(* Logix 5000 project; controller Comas_L4 vendor 1 type 14 code 193 rev 30.11; software revision 30.02; part 10 of 12 *)
(* tags used below, declared in another part *)
   Activation_Rouleau : BOOL;
   Axe_Codeur_Four : AXIS_CIP_DRIVE;
   Axe_Coupe_Fil : AXIS_CIP_DRIVE;
   Axe_Rouleaux_Canneles : AXIS_CIP_DRIVE;
   Axe_Virtuel_Coupe_Fil : AXIS_VIRTUAL;
   Axe_Virtuel_Maitre : AXIS_VIRTUAL;
   Cadencement_Moyennage_Codeur : FBD_TIMER;
   CAM_Virtuel_Coupe_Fil : CAM[100];
   CamGenerator_Coupe_Fil : AOI_CamGenerator_ST;
   CF_Mode_Came_Activation : BOOL;
   CF_Mode_Came_Engagement : BOOL;
   CF_Mode_Top_Activation : BOOL;
   CF_Mode_Top_Mouvement : BOOL;
   CO_Acquit_defaut : BOOL;
   CO_Activation : BOOL;
   CO_Axe_Codeur_Four_OK : BOOL;
   CO_Axe_Coupe_Fil_OK : BOOL;
   CO_Axe_Horizontal_Droit_OK : BOOL;
   CO_Axe_Horizontal_Gauche_OK : BOOL;
   CO_Axe_Pompe_Doseuse_OK : BOOL;
   CO_Axe_Rouleaux_Canneles_OK : BOOL;
   CO_Axe_Vertical_Droit_OK : BOOL;
   CO_Axe_Vertical_Gauche_OK : BOOL;
   CO_Consigne_Vitesse_Rouleaux : REAL;
   CO_Defaut_ARU_Armoire : BOOL;
   CO_Defaut_ARU_Machine : BOOL;
   CO_Defaut_ARU_Pupitre : BOOL;
   CO_Defaut_CamGenerator_Coupe_Fil : BOOL;
   CO_Defaut_CamGenerator_Horizontal : BOOL;
   CO_Defaut_CamGenerator_Vertical : BOOL;
   CO_Defaut_Clef_Graissage : BOOL;
   CO_Defaut_CPT_Porte1 : BOOL;
   CO_Defaut_CPT_Porte2 : BOOL;
   CO_Defaut_CPT_Porte3 : BOOL;
   CO_Defaut_CPT_Porte4 : BOOL;
   CO_Defaut_Eth_Codeur_Four : BOOL;
   CO_Defaut_Eth_Var_Coupe_Fil : BOOL;
   CO_Defaut_Eth_Var_H_Droit : BOOL;
   CO_Defaut_Eth_Var_H_Gauche : BOOL;
   CO_Defaut_Eth_Var_Pompe_Doseuse : BOOL;
   CO_Defaut_Eth_Var_Rouleaux : BOOL;
   CO_Defaut_Eth_Var_V_Droit : BOOL;
   CO_Defaut_Eth_Var_V_Gauche : BOOL;
   CO_Defaut_FDC : BOOL;
   CO_Defaut_FDC_Amont_Horizontal_Droit : BOOL;
   CO_Defaut_FDC_Amont_Horizontal_Gauche : BOOL;
   CO_Defaut_FDC_Aval_Horizontal_Droit : BOOL;
   CO_Defaut_FDC_Aval_Horizontal_Gauche : BOOL;
   CO_Defaut_FDC_Bas_Vertical_Droit : BOOL;
   CO_Defaut_FDC_Bas_Vertical_Gauche : BOOL;
   CO_Defaut_FDC_Coupe_Fil_Droit : BOOL;
   CO_Defaut_FDC_Coupe_Fil_Gauche : BOOL;
   CO_Defaut_FDC_Haut_Vertical_Droit : BOOL;
   CO_Defaut_FDC_Haut_Vertical_Gauche : BOOL;
   CO_Defaut_Four : BOOL;
   CO_Defaut_Presence_Coupe_Fil : BOOL;
   CO_Defaut_Relais_Securite : BOOL;
   CO_Defauts_Secondaires : BOOL;
   CO_Engage_Axe_Coupe_Fil : Engage_Axe;
   CO_Engage_Virtuel_Coupe_Fil : Engage_Axe_Virtuel;
   CO_Engagement : BOOL;
   CO_Engagement_Coupe_Fil : BOOL;
   CO_Ethernet_Code_Def_Codeur_Four : DINT;
   CO_Ethernet_Code_Def_Coupe_Fil : DINT;
   CO_Ethernet_Code_Def_H_Droit : DINT;
   CO_Ethernet_Code_Def_H_Gauche : DINT;
   CO_Ethernet_Code_Def_Pompe_Doseuse : DINT;
   CO_Ethernet_Code_Def_Rouleaux : DINT;
   CO_Ethernet_Code_Def_V_Droit : DINT;
   CO_Ethernet_Code_Def_V_Gauche : DINT;
   CO_Front_Activation : BOOL;
   CO_Init_Ok : BOOL;
   CO_Machine_sans_defaut : BOOL;
   CO_MAH_Virtuel_Coupe_Fil : MOTION_INSTRUCTION;
   CO_Pilotage_Coupe_Fil : Pilotage_Relatif_Virtuel;
   CO_Tempo_Valid_Recette : TIMER;
   CO_Top_Depart_Coupe_Fil : BOOL;
   CO_Top_Depart_Rouleaux : BOOL;
   CO_Validation_Recette : BOOL;
   ENT_CO_ARU_Armoire : ALIAS FOR Local:1:I.Pt03.Data;
   ENT_CO_ARU_Machine : ALIAS FOR Local:1:I.Pt05.Data;
   ENT_CO_ARU_Pupitre : ALIAS FOR Local:1:I.Pt04.Data;
   ENT_CO_BP_Rearmement : ALIAS FOR Local:1:I.Pt02.Data;
   ENT_CO_Clef_Graissage : ALIAS FOR Local:2:I.Pt02.Data;
   ENT_CO_CPT_Porte1 : ALIAS FOR Local:1:I.Pt06.Data;
   ENT_CO_CPT_Porte2 : ALIAS FOR Local:1:I.Pt07.Data;
   ENT_CO_CPT_Porte3 : ALIAS FOR Local:1:I.Pt08.Data;
   ENT_CO_CPT_Porte4 : ALIAS FOR Local:1:I.Pt09.Data;
   ENT_CO_FDC_Amont_Horizontal_Droit : ALIAS FOR Local:2:I.Pt15.Data;
   ENT_CO_FDC_Amont_Horizontal_Gauche : ALIAS FOR Local:2:I.Pt13.Data;
   ENT_CO_FDC_Aval_Horizontal_Droit : ALIAS FOR Local:2:I.Pt14.Data;
   ENT_CO_FDC_Aval_Horizontal_Gauche : ALIAS FOR Local:2:I.Pt12.Data;
   ENT_CO_FDC_Bas_Vertical_Droit : ALIAS FOR Local:2:I.Pt10.Data;
   ENT_CO_FDC_Bas_Vertical_Gauche : ALIAS FOR Local:2:I.Pt08.Data;
   ENT_CO_FDC_Coupe_Fil_Droit : BOOL;
   ENT_CO_FDC_Coupe_Fil_Gauche : BOOL;
   ENT_CO_FDC_Haut_Vertical_Droit : ALIAS FOR Local:2:I.Pt11.Data;
   ENT_CO_FDC_Haut_Vertical_Gauche : ALIAS FOR Local:2:I.Pt09.Data;
   ENT_CO_Relais_Securite : ALIAS FOR Local:1:I.Pt10.Data;
   ENT_Four_OK : ALIAS FOR Local:2:I.Pt01.Data;
   Front_Moyennage_Cadencement : FBD_ONESHOT;
   Front_Valid_Recette : BOOL;
   index_moyennage : DINT;
   Output_Cams_Coupe_Fil : Output_Cams;
   Output_Cams_Rouleaux : Output_Cams;
   PCAM_Coupe_Fil : UDT_CamGeneration;
   PCAM_Inter_PCAM_Coupe_Fil : CAM[100];
   Periode_Top_Depart_Coupe_FIl : REAL;
   RECETTE_CHAMP_VIDE : UDT_RECIPE;
   RECETTE_EC : UDT_RECIPE;
   RECETTE_HMI : UDT_HMI;
   RECETTE_SV : UDT_RECIPE[50];
   RSW_Acquit_defaut : BOOL;
   RSW_Depose_Active : BOOL;
   Speed_Control_Rouleaux : Axis_speed_control;
   Start_Cam_Logique_Rouleaux : REAL;
   Stop_Cam_Logique_Rouleaux : REAL;
   Tab_Moyennage_Codeur : REAL[200];
   Tab_Moyennage_Codeur_Temp : REAL[200];
   Tempo_Off_Arret_Rouleaux : TIMER;
   Temporisation_Engagement_Virtuel_CF : TIMER;
   Vitesse_Codeur : REAL;
   Vitesse_Mini_Coupe_Fil : REAL;
   Vitesse_Moy_Codeur : REAL;
   Vitesse_Moy_Temp : REAL;
(* Comas, continued *)

ROUTINE F02_Engagement_Coupe_Fil   (* ladder *)
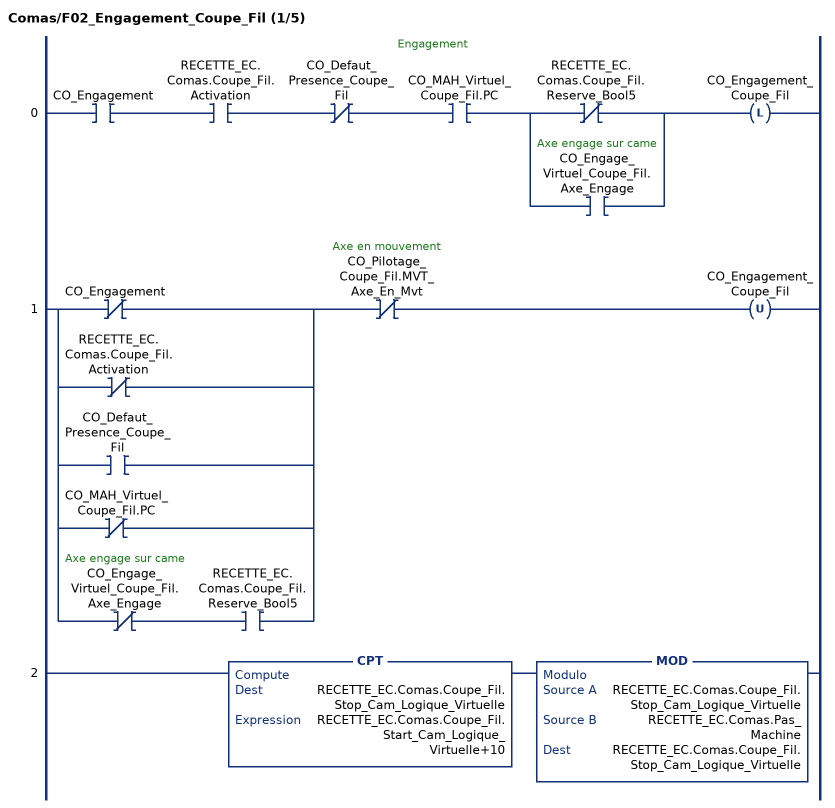
   // Engagement
   0: XIC(CO_Engagement)XIC(RECETTE_EC.Comas.Coupe_Fil.Activation)XIO(CO_Defaut_Presence_Coupe_Fil)XIC(CO_MAH_Virtuel_Coupe_Fil.PC)[XIO(RECETTE_EC.Comas.Coupe_Fil.Reserve_Bool5) ,XIC(CO_Engage_Virtuel_Coupe_Fil.Axe_Engage) ]OTL(CO_Engagement_Coupe_Fil);
   1: [XIO(CO_Engagement) ,XIO(RECETTE_EC.Comas.Coupe_Fil.Activation) ,XIC(CO_Defaut_Presence_Coupe_Fil) ,XIO(CO_MAH_Virtuel_Coupe_Fil.PC) ,XIO(CO_Engage_Virtuel_Coupe_Fil.Axe_Engage) XIC(RECETTE_EC.Comas.Coupe_Fil.Reserve_Bool5) ]XIO(CO_Pilotage_Coupe_Fil.MVT_Axe_En_Mvt)OTU(CO_Engagement_Coupe_Fil);
   2: CPT(RECETTE_EC.Comas.Coupe_Fil.Stop_Cam_Logique_Virtuelle,RECETTE_EC.Comas.Coupe_Fil.Start_Cam_Logique_Virtuelle+10)MOD(RECETTE_EC.Comas.Coupe_Fil.Stop_Cam_Logique_Virtuelle,RECETTE_EC.Comas.Pas_Machine,RECETTE_EC.Comas.Coupe_Fil.Stop_Cam_Logique_Virtuelle);
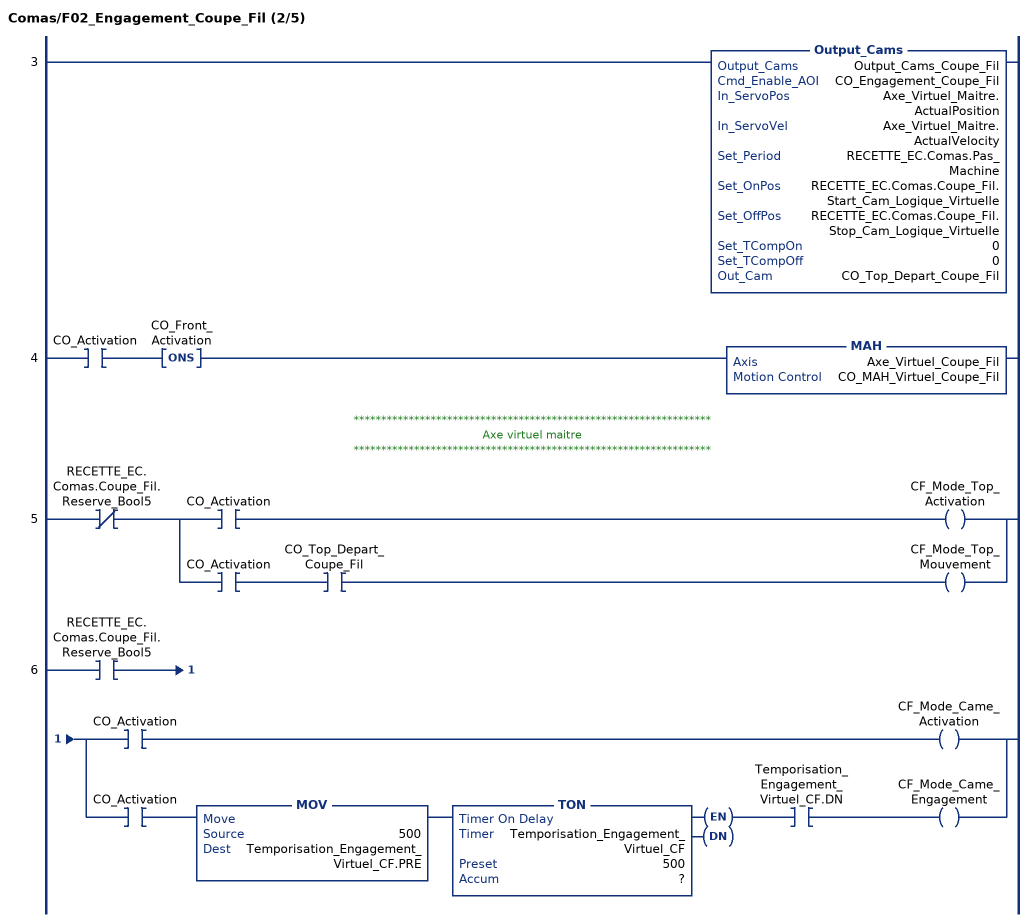
   3: Output_Cams(Output_Cams_Coupe_Fil,CO_Engagement_Coupe_Fil,Axe_Virtuel_Maitre.ActualPosition,Axe_Virtuel_Maitre.ActualVelocity,RECETTE_EC.Comas.Pas_Machine,RECETTE_EC.Comas.Coupe_Fil.Start_Cam_Logique_Virtuelle,RECETTE_EC.Comas.Coupe_Fil.Stop_Cam_Logique_Virtuelle,0,0,CO_Top_Depart_Coupe_Fil);
   4: XIC(CO_Activation)ONS(CO_Front_Activation)MAH(Axe_Virtuel_Coupe_Fil,CO_MAH_Virtuel_Coupe_Fil);
   // *****************************************************************
   // Axe virtuel maitre
   // *****************************************************************
   5: XIO(RECETTE_EC.Comas.Coupe_Fil.Reserve_Bool5)[XIC(CO_Activation) OTE(CF_Mode_Top_Activation) ,XIC(CO_Activation) XIC(CO_Top_Depart_Coupe_Fil) OTE(CF_Mode_Top_Mouvement) ];
   6: XIC(RECETTE_EC.Comas.Coupe_Fil.Reserve_Bool5)[XIC(CO_Activation) OTE(CF_Mode_Came_Activation) ,XIC(CO_Activation) MOV(500,Temporisation_Engagement_Virtuel_CF.PRE) TON(Temporisation_Engagement_Virtuel_CF,?,?) XIC(Temporisation_Engagement_Virtuel_CF.DN) OTE(CF_Mode_Came_Engagement) ];
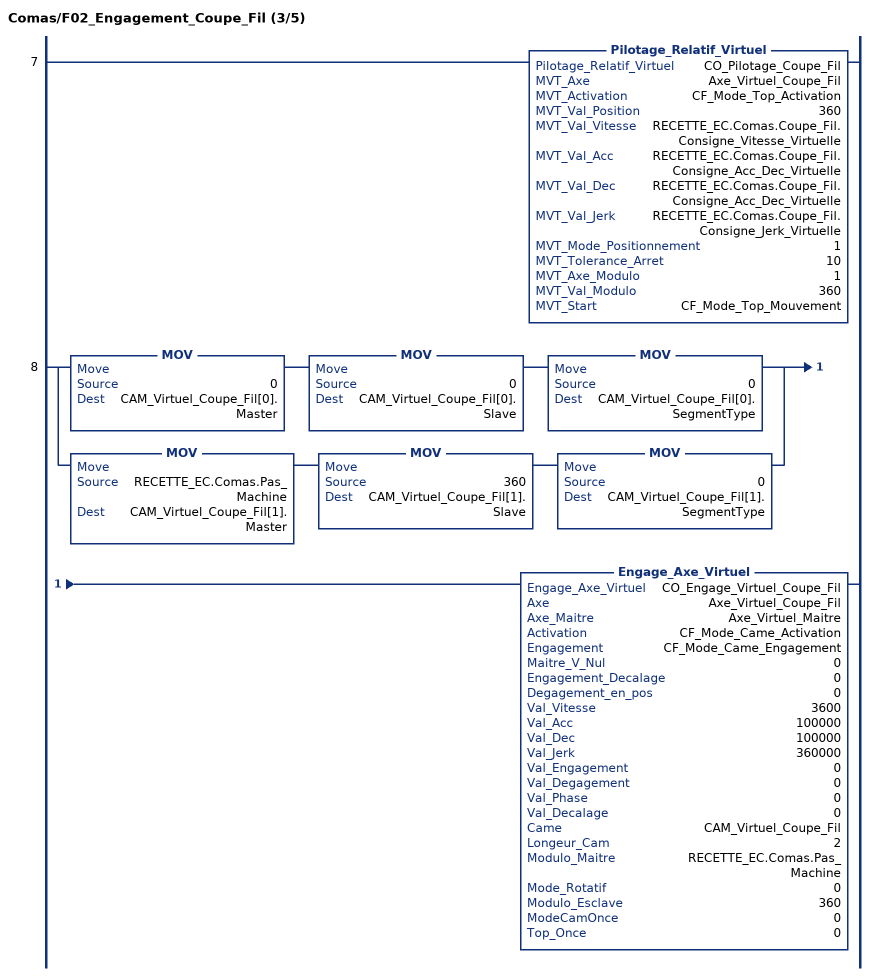
   7: Pilotage_Relatif_Virtuel(CO_Pilotage_Coupe_Fil,Axe_Virtuel_Coupe_Fil,CF_Mode_Top_Activation,360,RECETTE_EC.Comas.Coupe_Fil.Consigne_Vitesse_Virtuelle,RECETTE_EC.Comas.Coupe_Fil.Consigne_Acc_Dec_Virtuelle,RECETTE_EC.Comas.Coupe_Fil.Consigne_Acc_Dec_Virtuelle,RECETTE_EC.Comas.Coupe_Fil.Consigne_Jerk_Virtuelle,1,10,1,360,CF_Mode_Top_Mouvement);
   8: [MOV(0,CAM_Virtuel_Coupe_Fil[0].Master) MOV(0,CAM_Virtuel_Coupe_Fil[0].Slave) MOV(0,CAM_Virtuel_Coupe_Fil[0].SegmentType) ,MOV(RECETTE_EC.Comas.Pas_Machine,CAM_Virtuel_Coupe_Fil[1].Master) MOV(360,CAM_Virtuel_Coupe_Fil[1].Slave) MOV(0,CAM_Virtuel_Coupe_Fil[1].SegmentType) ]Engage_Axe_Virtuel(CO_Engage_Virtuel_Coupe_Fil,Axe_Virtuel_Coupe_Fil,Axe_Virtuel_Maitre,CF_Mode_Came_Activation,CF_Mode_Came_Engagement,0,0,0,3600,100000,100000,360000,0,0,0,0,CAM_Virtuel_Coupe_Fil,2,RECETTE_EC.Comas.Pas_Machine,0,360,0,0);
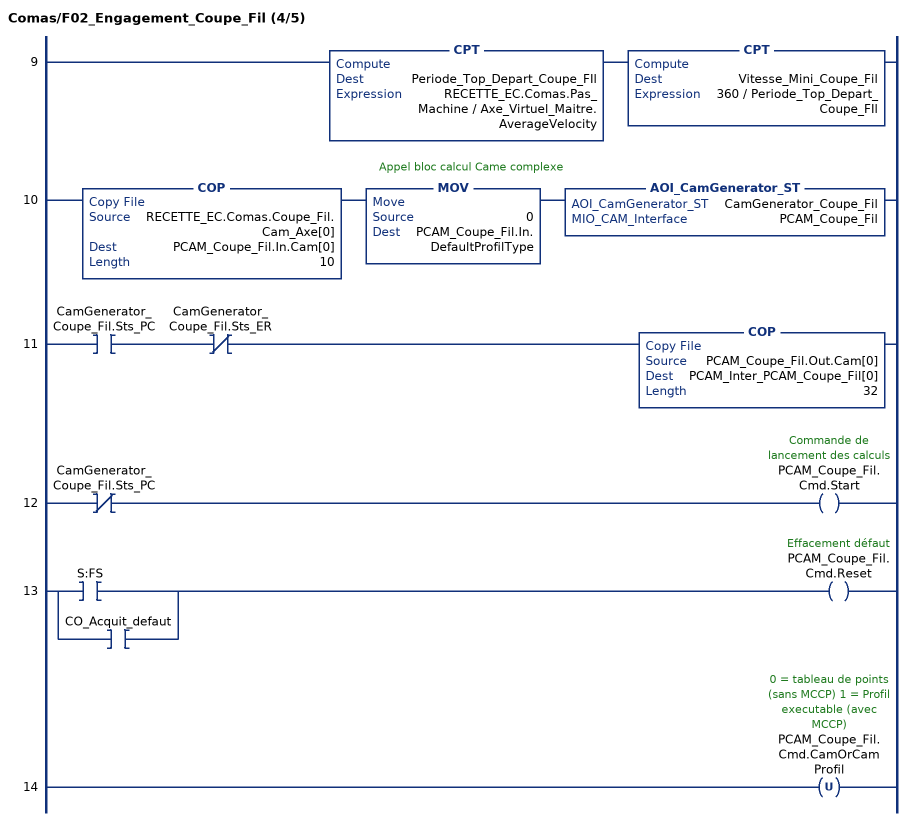
   9: CPT(Periode_Top_Depart_Coupe_FIl,RECETTE_EC.Comas.Pas_Machine / Axe_Virtuel_Maitre.AverageVelocity)CPT(Vitesse_Mini_Coupe_Fil,360 / Periode_Top_Depart_Coupe_FIl);
   // Appel bloc calcul Came complexe
   10: COP(RECETTE_EC.Comas.Coupe_Fil.Cam_Axe[0],PCAM_Coupe_Fil.In.Cam[0],10)MOV(0,PCAM_Coupe_Fil.In.DefaultProfilType)AOI_CamGenerator_ST(CamGenerator_Coupe_Fil,PCAM_Coupe_Fil);
   11: XIC(CamGenerator_Coupe_Fil.Sts_PC)XIO(CamGenerator_Coupe_Fil.Sts_ER)COP(PCAM_Coupe_Fil.Out.Cam[0],PCAM_Inter_PCAM_Coupe_Fil[0],32);
   12: XIO(CamGenerator_Coupe_Fil.Sts_PC)OTE(PCAM_Coupe_Fil.Cmd.Start);
   13: [XIC(S:FS) ,XIC(CO_Acquit_defaut) ]OTE(PCAM_Coupe_Fil.Cmd.Reset);
   14: OTU(PCAM_Coupe_Fil.Cmd.CamOrCamProfil);
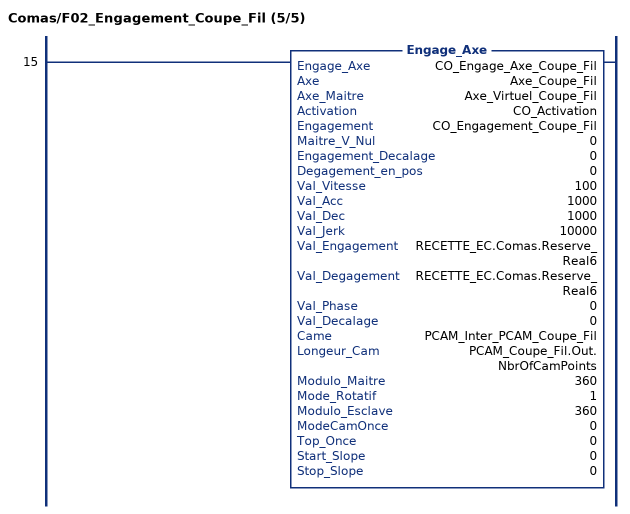
   15: Engage_Axe(CO_Engage_Axe_Coupe_Fil,Axe_Coupe_Fil,Axe_Virtuel_Coupe_Fil,CO_Activation,CO_Engagement_Coupe_Fil,0,0,0,100,1000,1000,10000,RECETTE_EC.Comas.Reserve_Real6,RECETTE_EC.Comas.Reserve_Real6,0,0,PCAM_Inter_PCAM_Coupe_Fil,PCAM_Coupe_Fil.Out.NbrOfCamPoints,360,1,360,0,0,0,0);
END_ROUTINE

ROUTINE F03_Engagement_Rouleaux   (* ladder *)
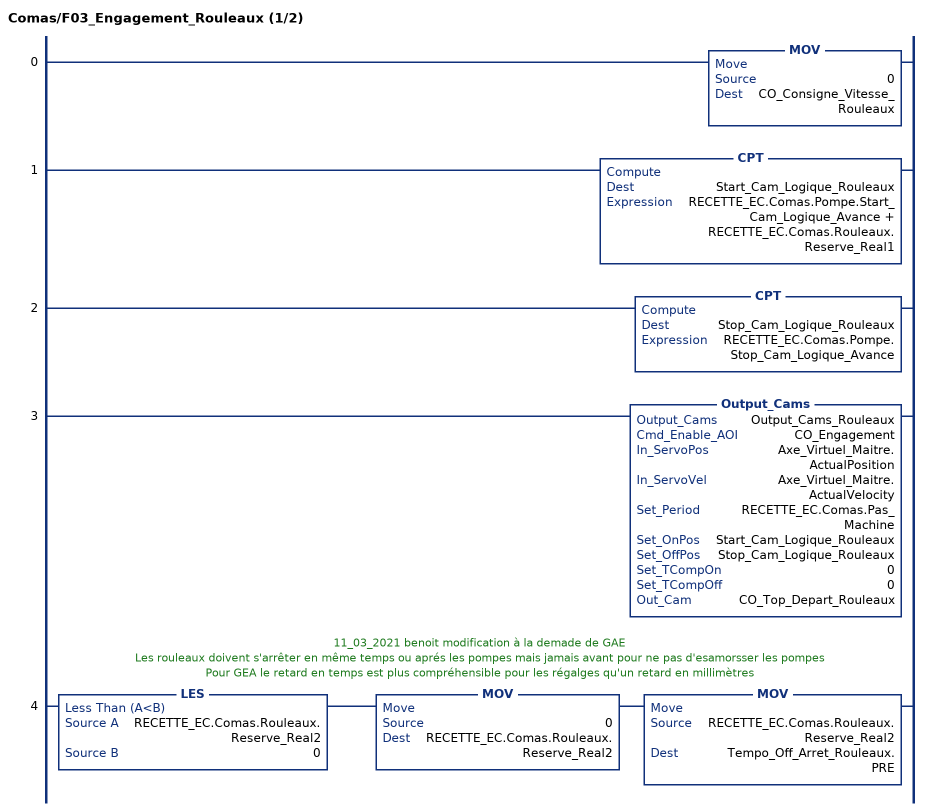
   0: MOV(0,CO_Consigne_Vitesse_Rouleaux);
   1: CPT(Start_Cam_Logique_Rouleaux,RECETTE_EC.Comas.Pompe.Start_Cam_Logique_Avance + RECETTE_EC.Comas.Rouleaux.Reserve_Real1);
   2: CPT(Stop_Cam_Logique_Rouleaux,RECETTE_EC.Comas.Pompe.Stop_Cam_Logique_Avance);
   3: Output_Cams(Output_Cams_Rouleaux,CO_Engagement,Axe_Virtuel_Maitre.ActualPosition,Axe_Virtuel_Maitre.ActualVelocity,RECETTE_EC.Comas.Pas_Machine,Start_Cam_Logique_Rouleaux,Stop_Cam_Logique_Rouleaux,0,0,CO_Top_Depart_Rouleaux);
   // 11_03_2021 benoit modification à la demade de GAE
   // Les rouleaux doivent s'arrêter en même temps ou aprés les pompes mais jamais avant pour ne pas d'esamorsser les pompes
   // Pour GEA le retard en temps est plus compréhensible pour les régalges qu'un retard en millimètres
   4: LES(RECETTE_EC.Comas.Rouleaux.Reserve_Real2,0)MOV(0,RECETTE_EC.Comas.Rouleaux.Reserve_Real2)MOV(RECETTE_EC.Comas.Rouleaux.Reserve_Real2,Tempo_Off_Arret_Rouleaux.PRE);
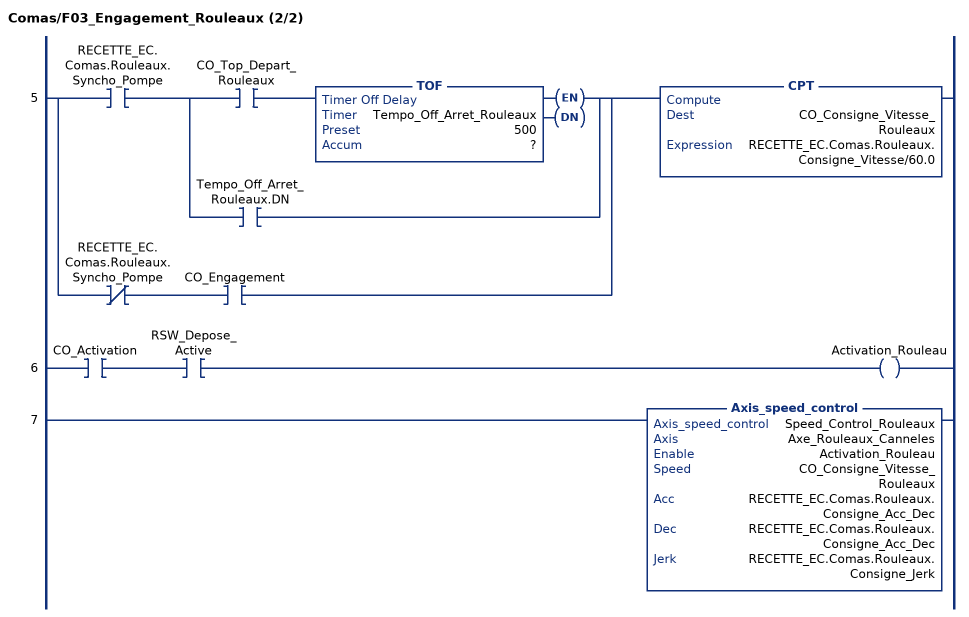
   5: [XIC(RECETTE_EC.Comas.Rouleaux.Syncho_Pompe) [XIC(CO_Top_Depart_Rouleaux) TOF(Tempo_Off_Arret_Rouleaux,?,?) ,XIC(Tempo_Off_Arret_Rouleaux.DN) ] ,XIO(RECETTE_EC.Comas.Rouleaux.Syncho_Pompe) XIC(CO_Engagement) ]CPT(CO_Consigne_Vitesse_Rouleaux,RECETTE_EC.Comas.Rouleaux.Consigne_Vitesse/60.0);
   6: XIC(CO_Activation)XIC(RSW_Depose_Active)OTE(Activation_Rouleau);
   7: Axis_speed_control(Speed_Control_Rouleaux,Axe_Rouleaux_Canneles,Activation_Rouleau,CO_Consigne_Vitesse_Rouleaux,RECETTE_EC.Comas.Rouleaux.Consigne_Acc_Dec,RECETTE_EC.Comas.Rouleaux.Consigne_Acc_Dec,RECETTE_EC.Comas.Rouleaux.Consigne_Jerk);
END_ROUTINE

ROUTINE F05_Moyennage_Codeur   (* structured text *)
   // Codeur
   Vitesse_Codeur:=Axe_Codeur_Four.AverageVelocity;
   
   // Cadencement
   Cadencement_Moyennage_Codeur.PRE := 1000;
   Cadencement_Moyennage_Codeur.Reset := Cadencement_Moyennage_Codeur.DN;
   Cadencement_Moyennage_Codeur.TimerEnable := NOT Cadencement_Moyennage_Codeur.DN;
   TONR(Cadencement_Moyennage_Codeur);
   
   Front_Moyennage_Cadencement.InputBit:=Cadencement_Moyennage_Codeur.DN;
   OSRI(Front_Moyennage_Cadencement);
   
   // Decalage Tableau
   IF Front_Moyennage_Cadencement.OutputBit THEN
   	Tab_Moyennage_Codeur[0]:=Vitesse_Codeur;
   	COP(Tab_Moyennage_Codeur[0],Tab_Moyennage_Codeur_Temp[1],190);
   	COP(Tab_Moyennage_Codeur_Temp[0],Tab_Moyennage_Codeur[0],190);
   END_IF;
   Vitesse_Moy_Temp:=0;
   FOR index_moyennage:=1 TO 150 BY 1 DO
   	Vitesse_Moy_Temp:=Vitesse_Moy_Temp+Tab_Moyennage_Codeur[index_moyennage];
   END_FOR;
   Vitesse_Moy_Codeur:=Vitesse_Moy_Temp/150;
   
   
   
   
   
   
   
   
   
   
   
   
   
   
   
   
   
   
END_ROUTINE
END_PROGRAM

PROGRAM General   (* main routine A00_Princ *)

ROUTINE A00_Princ   (* ladder *)
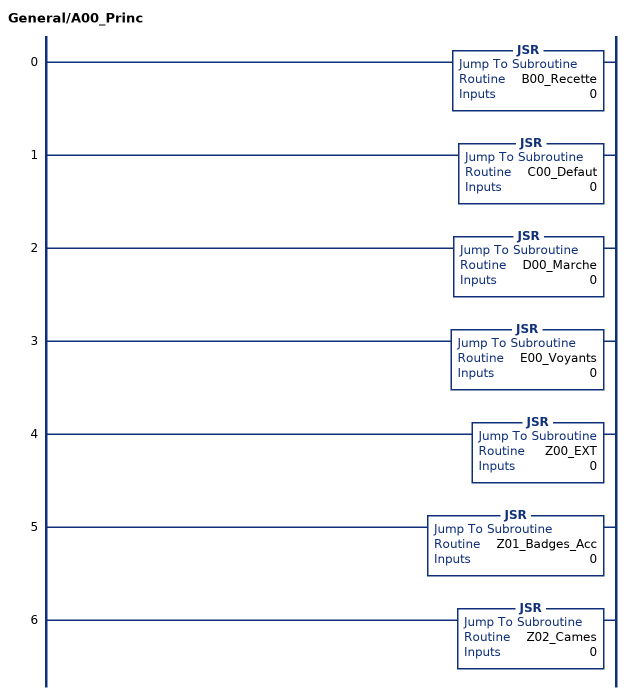
   0: JSR(B00_Recette,0);
   1: JSR(C00_Defaut,0);
   2: JSR(D00_Marche,0);
   3: JSR(E00_Voyants,0);
   4: JSR(Z00_EXT,0);
   5: JSR(Z01_Badges_Acc,0);
   6: JSR(Z02_Cames,0);
END_ROUTINE

ROUTINE B00_Recette   (* ladder *)
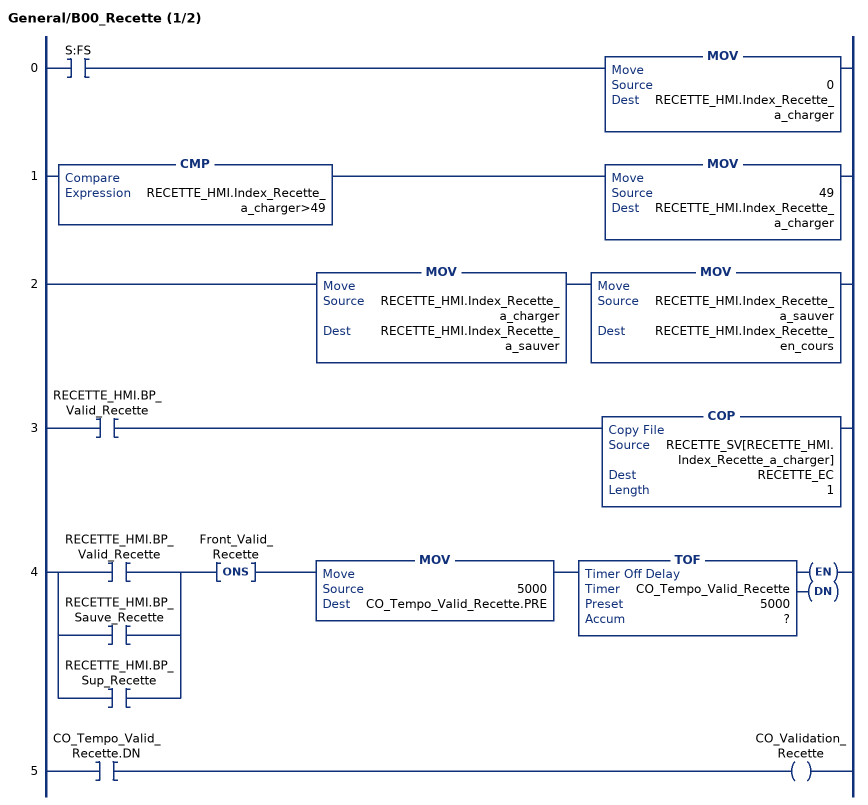
   0: XIC(S:FS)MOV(0,RECETTE_HMI.Index_Recette_a_charger);
   1: CMP(RECETTE_HMI.Index_Recette_a_charger>49)MOV(49,RECETTE_HMI.Index_Recette_a_charger);
   2: MOV(RECETTE_HMI.Index_Recette_a_charger,RECETTE_HMI.Index_Recette_a_sauver)MOV(RECETTE_HMI.Index_Recette_a_sauver,RECETTE_HMI.Index_Recette_en_cours);
   3: XIC(RECETTE_HMI.BP_Valid_Recette)COP(RECETTE_SV[RECETTE_HMI.Index_Recette_a_charger],RECETTE_EC,1);
   4: [XIC(RECETTE_HMI.BP_Valid_Recette) ,XIC(RECETTE_HMI.BP_Sauve_Recette) ,XIC(RECETTE_HMI.BP_Sup_Recette) ]ONS(Front_Valid_Recette)MOV(5000,CO_Tempo_Valid_Recette.PRE)TOF(CO_Tempo_Valid_Recette,?,?);
   5: XIC(CO_Tempo_Valid_Recette.DN)OTE(CO_Validation_Recette);
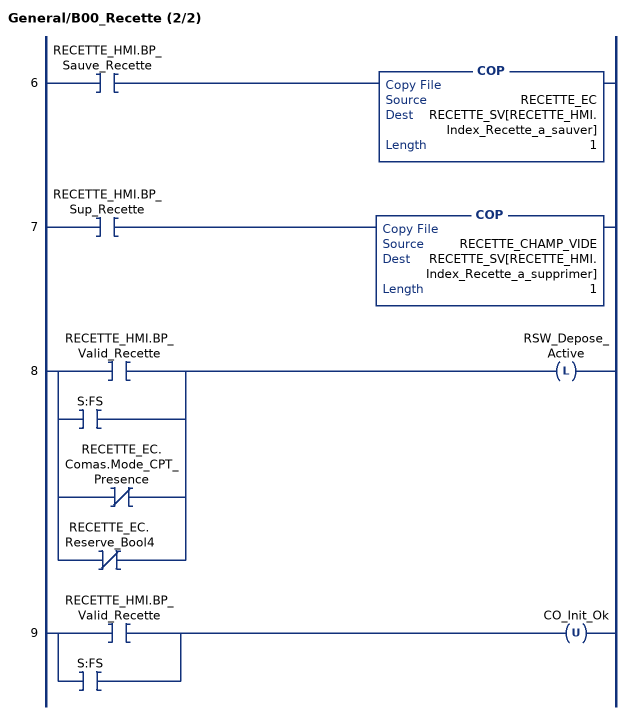
   6: XIC(RECETTE_HMI.BP_Sauve_Recette)COP(RECETTE_EC,RECETTE_SV[RECETTE_HMI.Index_Recette_a_sauver],1);
   7: XIC(RECETTE_HMI.BP_Sup_Recette)COP(RECETTE_CHAMP_VIDE,RECETTE_SV[RECETTE_HMI.Index_Recette_a_supprimer],1);
   8: [XIC(RECETTE_HMI.BP_Valid_Recette) ,XIC(S:FS) ,XIO(RECETTE_EC.Comas.Mode_CPT_Presence) ,XIO(RECETTE_EC.Reserve_Bool4) ]OTL(RSW_Depose_Active);
   9: [XIC(RECETTE_HMI.BP_Valid_Recette) ,XIC(S:FS) ]OTU(CO_Init_Ok);
END_ROUTINE

ROUTINE C00_Defaut   (* ladder *)
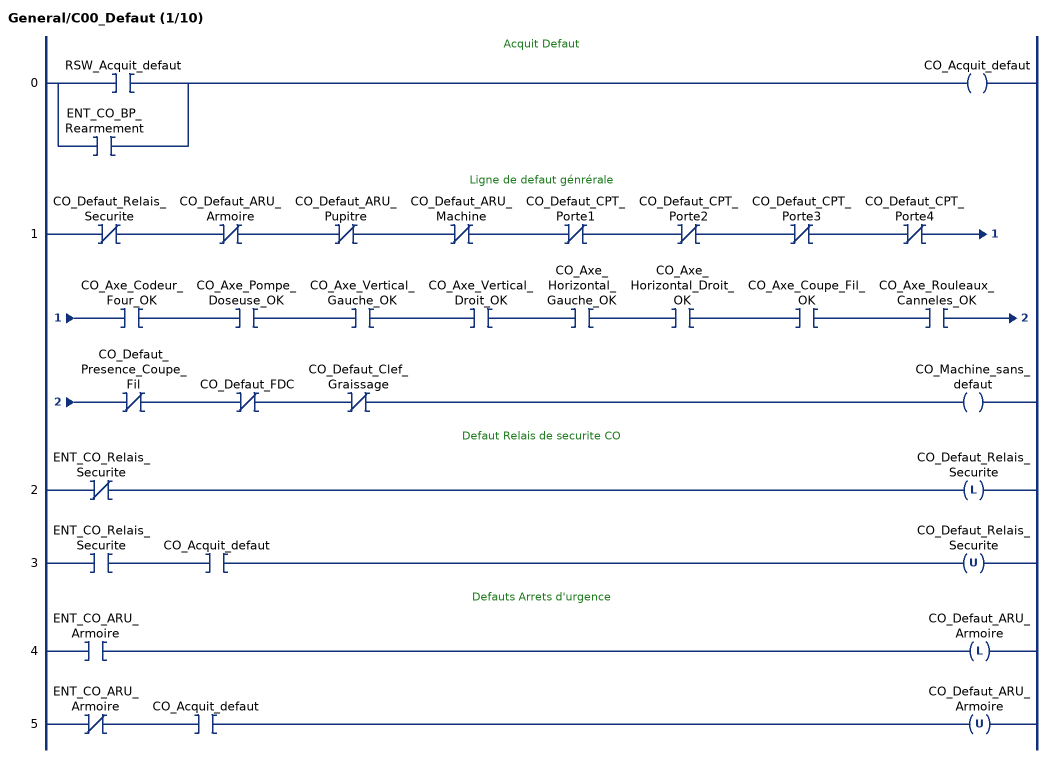
   // Acquit Defaut
   0: [XIC(RSW_Acquit_defaut) ,XIC(ENT_CO_BP_Rearmement) ]OTE(CO_Acquit_defaut);
   // Ligne de defaut génrérale
   1: XIO(CO_Defaut_Relais_Securite)XIO(CO_Defaut_ARU_Armoire)XIO(CO_Defaut_ARU_Pupitre)XIO(CO_Defaut_ARU_Machine)XIO(CO_Defaut_CPT_Porte1)XIO(CO_Defaut_CPT_Porte2)XIO(CO_Defaut_CPT_Porte3)XIO(CO_Defaut_CPT_Porte4)XIC(CO_Axe_Codeur_Four_OK)XIC(CO_Axe_Pompe_Doseuse_OK)XIC(CO_Axe_Vertical_Gauche_OK)XIC(CO_Axe_Vertical_Droit_OK)XIC(CO_Axe_Horizontal_Gauche_OK)XIC(CO_Axe_Horizontal_Droit_OK)XIC(CO_Axe_Coupe_Fil_OK)XIC(CO_Axe_Rouleaux_Canneles_OK)XIO(CO_Defaut_Presence_Coupe_Fil)XIO(CO_Defaut_FDC)XIO(CO_Defaut_Clef_Graissage)OTE(CO_Machine_sans_defaut);
   // Defaut Relais de securite CO
   2: XIO(ENT_CO_Relais_Securite)OTL(CO_Defaut_Relais_Securite);
   3: XIC(ENT_CO_Relais_Securite)XIC(CO_Acquit_defaut)OTU(CO_Defaut_Relais_Securite);
   // Defauts Arrets d'urgence
   4: XIC(ENT_CO_ARU_Armoire)OTL(CO_Defaut_ARU_Armoire);
   5: XIO(ENT_CO_ARU_Armoire)XIC(CO_Acquit_defaut)OTU(CO_Defaut_ARU_Armoire);
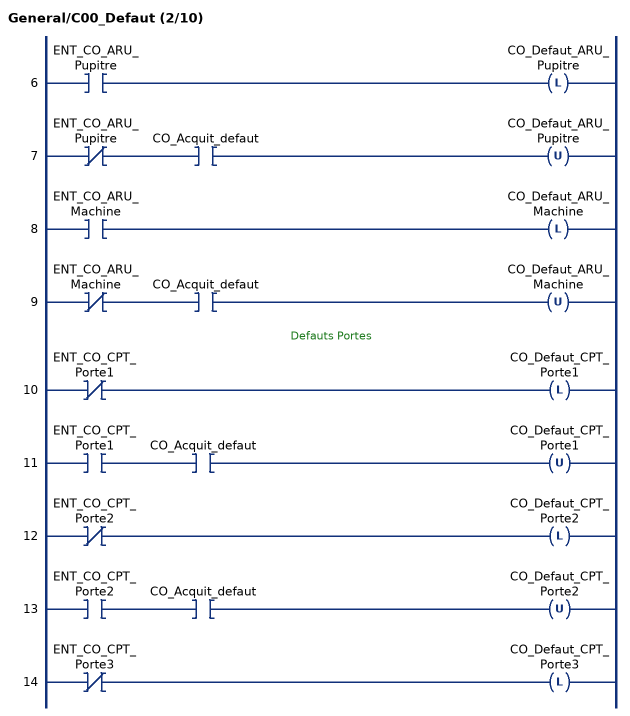
   6: XIC(ENT_CO_ARU_Pupitre)OTL(CO_Defaut_ARU_Pupitre);
   7: XIO(ENT_CO_ARU_Pupitre)XIC(CO_Acquit_defaut)OTU(CO_Defaut_ARU_Pupitre);
   8: XIC(ENT_CO_ARU_Machine)OTL(CO_Defaut_ARU_Machine);
   9: XIO(ENT_CO_ARU_Machine)XIC(CO_Acquit_defaut)OTU(CO_Defaut_ARU_Machine);
   // Defauts Portes
   10: XIO(ENT_CO_CPT_Porte1)OTL(CO_Defaut_CPT_Porte1);
   11: XIC(ENT_CO_CPT_Porte1)XIC(CO_Acquit_defaut)OTU(CO_Defaut_CPT_Porte1);
   12: XIO(ENT_CO_CPT_Porte2)OTL(CO_Defaut_CPT_Porte2);
   13: XIC(ENT_CO_CPT_Porte2)XIC(CO_Acquit_defaut)OTU(CO_Defaut_CPT_Porte2);
   14: XIO(ENT_CO_CPT_Porte3)OTL(CO_Defaut_CPT_Porte3);
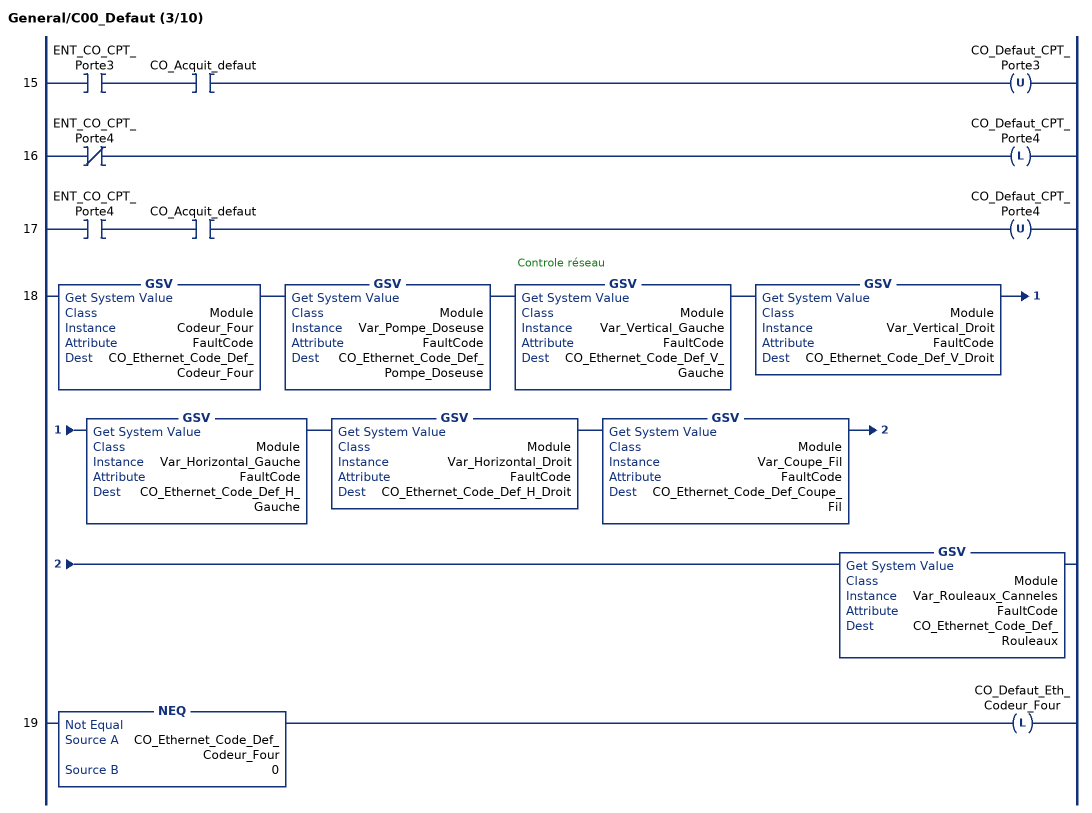
   15: XIC(ENT_CO_CPT_Porte3)XIC(CO_Acquit_defaut)OTU(CO_Defaut_CPT_Porte3);
   16: XIO(ENT_CO_CPT_Porte4)OTL(CO_Defaut_CPT_Porte4);
   17: XIC(ENT_CO_CPT_Porte4)XIC(CO_Acquit_defaut)OTU(CO_Defaut_CPT_Porte4);
   // Controle réseau
   18: GSV(Module,Codeur_Four,FaultCode,CO_Ethernet_Code_Def_Codeur_Four)GSV(Module,Var_Pompe_Doseuse,FaultCode,CO_Ethernet_Code_Def_Pompe_Doseuse)GSV(Module,Var_Vertical_Gauche,FaultCode,CO_Ethernet_Code_Def_V_Gauche)GSV(Module,Var_Vertical_Droit,FaultCode,CO_Ethernet_Code_Def_V_Droit)GSV(Module,Var_Horizontal_Gauche,FaultCode,CO_Ethernet_Code_Def_H_Gauche)GSV(Module,Var_Horizontal_Droit,FaultCode,CO_Ethernet_Code_Def_H_Droit)GSV(Module,Var_Coupe_Fil,FaultCode,CO_Ethernet_Code_Def_Coupe_Fil)GSV(Module,Var_Rouleaux_Canneles,FaultCode,CO_Ethernet_Code_Def_Rouleaux);
   19: NEQ(CO_Ethernet_Code_Def_Codeur_Four,0)OTL(CO_Defaut_Eth_Codeur_Four);
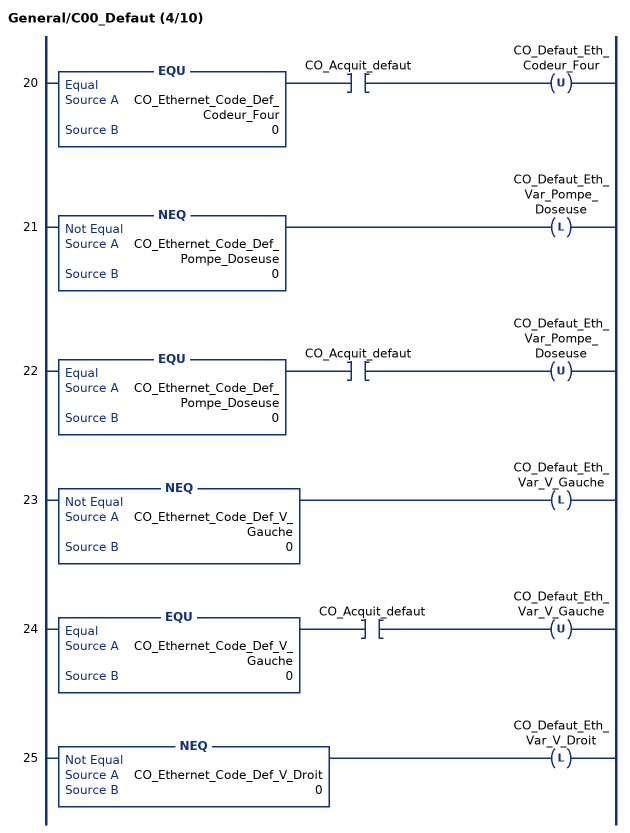
   20: EQU(CO_Ethernet_Code_Def_Codeur_Four,0)XIC(CO_Acquit_defaut)OTU(CO_Defaut_Eth_Codeur_Four);
   21: NEQ(CO_Ethernet_Code_Def_Pompe_Doseuse,0)OTL(CO_Defaut_Eth_Var_Pompe_Doseuse);
   22: EQU(CO_Ethernet_Code_Def_Pompe_Doseuse,0)XIC(CO_Acquit_defaut)OTU(CO_Defaut_Eth_Var_Pompe_Doseuse);
   23: NEQ(CO_Ethernet_Code_Def_V_Gauche,0)OTL(CO_Defaut_Eth_Var_V_Gauche);
   24: EQU(CO_Ethernet_Code_Def_V_Gauche,0)XIC(CO_Acquit_defaut)OTU(CO_Defaut_Eth_Var_V_Gauche);
   25: NEQ(CO_Ethernet_Code_Def_V_Droit,0)OTL(CO_Defaut_Eth_Var_V_Droit);
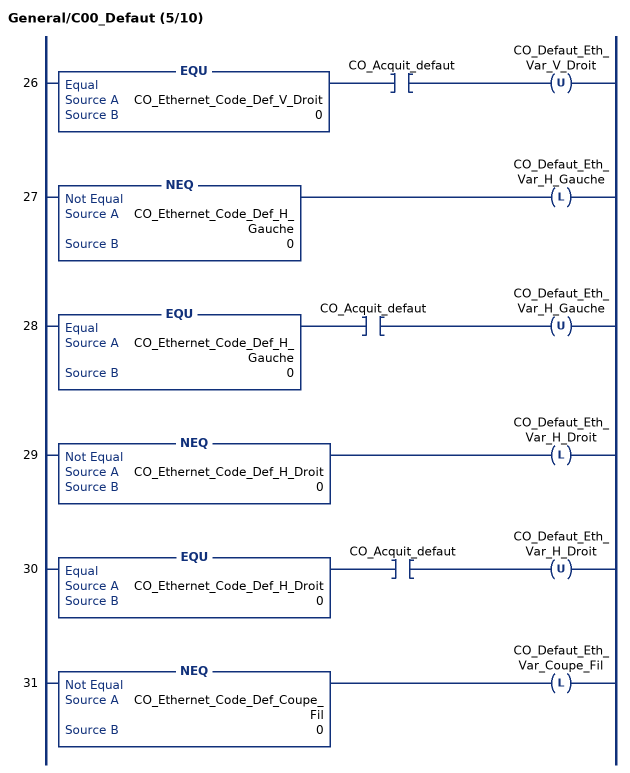
   26: EQU(CO_Ethernet_Code_Def_V_Droit,0)XIC(CO_Acquit_defaut)OTU(CO_Defaut_Eth_Var_V_Droit);
   27: NEQ(CO_Ethernet_Code_Def_H_Gauche,0)OTL(CO_Defaut_Eth_Var_H_Gauche);
   28: EQU(CO_Ethernet_Code_Def_H_Gauche,0)XIC(CO_Acquit_defaut)OTU(CO_Defaut_Eth_Var_H_Gauche);
   29: NEQ(CO_Ethernet_Code_Def_H_Droit,0)OTL(CO_Defaut_Eth_Var_H_Droit);
   30: EQU(CO_Ethernet_Code_Def_H_Droit,0)XIC(CO_Acquit_defaut)OTU(CO_Defaut_Eth_Var_H_Droit);
   31: NEQ(CO_Ethernet_Code_Def_Coupe_Fil,0)OTL(CO_Defaut_Eth_Var_Coupe_Fil);
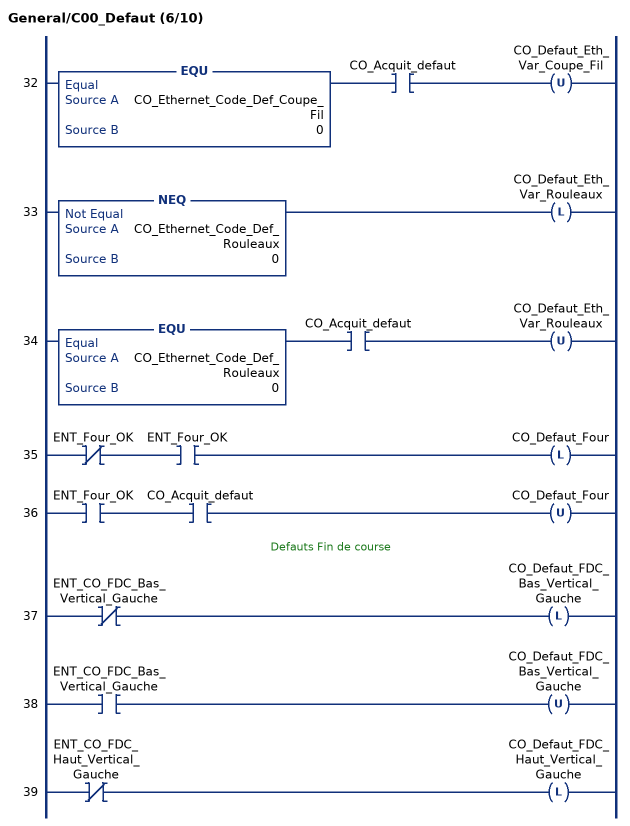
   32: EQU(CO_Ethernet_Code_Def_Coupe_Fil,0)XIC(CO_Acquit_defaut)OTU(CO_Defaut_Eth_Var_Coupe_Fil);
   33: NEQ(CO_Ethernet_Code_Def_Rouleaux,0)OTL(CO_Defaut_Eth_Var_Rouleaux);
   34: EQU(CO_Ethernet_Code_Def_Rouleaux,0)XIC(CO_Acquit_defaut)OTU(CO_Defaut_Eth_Var_Rouleaux);
   35: XIO(ENT_Four_OK)XIC(ENT_Four_OK)OTL(CO_Defaut_Four);
   36: XIC(ENT_Four_OK)XIC(CO_Acquit_defaut)OTU(CO_Defaut_Four);
   // Defauts Fin de course
   37: XIO(ENT_CO_FDC_Bas_Vertical_Gauche)OTL(CO_Defaut_FDC_Bas_Vertical_Gauche);
   38: XIC(ENT_CO_FDC_Bas_Vertical_Gauche)OTU(CO_Defaut_FDC_Bas_Vertical_Gauche);
   39: XIO(ENT_CO_FDC_Haut_Vertical_Gauche)OTL(CO_Defaut_FDC_Haut_Vertical_Gauche);
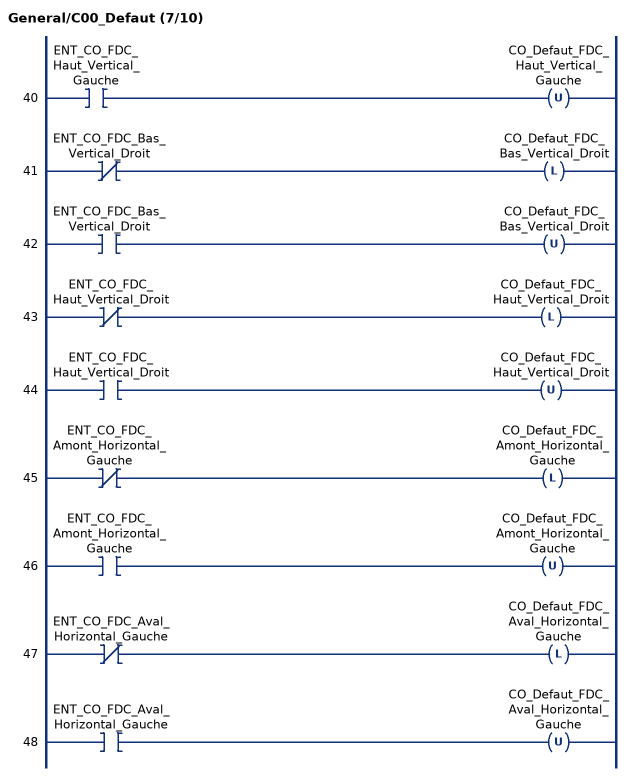
   40: XIC(ENT_CO_FDC_Haut_Vertical_Gauche)OTU(CO_Defaut_FDC_Haut_Vertical_Gauche);
   41: XIO(ENT_CO_FDC_Bas_Vertical_Droit)OTL(CO_Defaut_FDC_Bas_Vertical_Droit);
   42: XIC(ENT_CO_FDC_Bas_Vertical_Droit)OTU(CO_Defaut_FDC_Bas_Vertical_Droit);
   43: XIO(ENT_CO_FDC_Haut_Vertical_Droit)OTL(CO_Defaut_FDC_Haut_Vertical_Droit);
   44: XIC(ENT_CO_FDC_Haut_Vertical_Droit)OTU(CO_Defaut_FDC_Haut_Vertical_Droit);
   45: XIO(ENT_CO_FDC_Amont_Horizontal_Gauche)OTL(CO_Defaut_FDC_Amont_Horizontal_Gauche);
   46: XIC(ENT_CO_FDC_Amont_Horizontal_Gauche)OTU(CO_Defaut_FDC_Amont_Horizontal_Gauche);
   47: XIO(ENT_CO_FDC_Aval_Horizontal_Gauche)OTL(CO_Defaut_FDC_Aval_Horizontal_Gauche);
   48: XIC(ENT_CO_FDC_Aval_Horizontal_Gauche)OTU(CO_Defaut_FDC_Aval_Horizontal_Gauche);
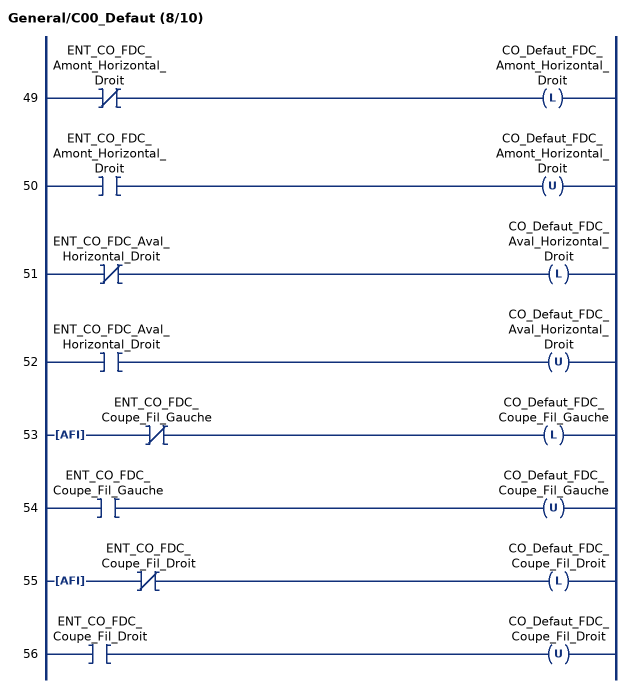
   49: XIO(ENT_CO_FDC_Amont_Horizontal_Droit)OTL(CO_Defaut_FDC_Amont_Horizontal_Droit);
   50: XIC(ENT_CO_FDC_Amont_Horizontal_Droit)OTU(CO_Defaut_FDC_Amont_Horizontal_Droit);
   51: XIO(ENT_CO_FDC_Aval_Horizontal_Droit)OTL(CO_Defaut_FDC_Aval_Horizontal_Droit);
   52: XIC(ENT_CO_FDC_Aval_Horizontal_Droit)OTU(CO_Defaut_FDC_Aval_Horizontal_Droit);
   53: AFI()XIO(ENT_CO_FDC_Coupe_Fil_Gauche)OTL(CO_Defaut_FDC_Coupe_Fil_Gauche);
   54: XIC(ENT_CO_FDC_Coupe_Fil_Gauche)OTU(CO_Defaut_FDC_Coupe_Fil_Gauche);
   55: AFI()XIO(ENT_CO_FDC_Coupe_Fil_Droit)OTL(CO_Defaut_FDC_Coupe_Fil_Droit);
   56: XIC(ENT_CO_FDC_Coupe_Fil_Droit)OTU(CO_Defaut_FDC_Coupe_Fil_Droit);
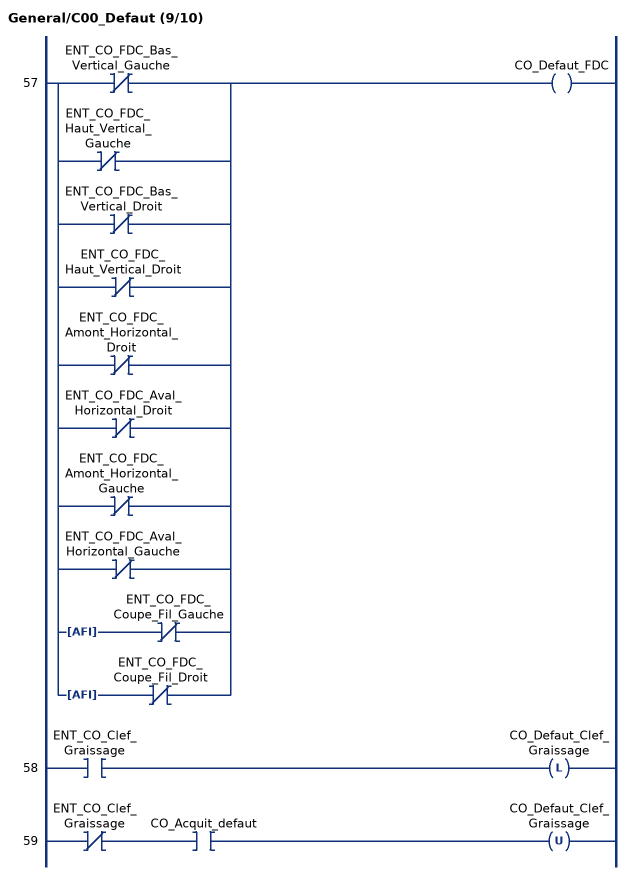
   57: [XIO(ENT_CO_FDC_Bas_Vertical_Gauche) ,XIO(ENT_CO_FDC_Haut_Vertical_Gauche) ,XIO(ENT_CO_FDC_Bas_Vertical_Droit) ,XIO(ENT_CO_FDC_Haut_Vertical_Droit) ,XIO(ENT_CO_FDC_Amont_Horizontal_Droit) ,XIO(ENT_CO_FDC_Aval_Horizontal_Droit) ,XIO(ENT_CO_FDC_Amont_Horizontal_Gauche) ,XIO(ENT_CO_FDC_Aval_Horizontal_Gauche) ,AFI() XIO(ENT_CO_FDC_Coupe_Fil_Gauche) ,AFI() XIO(ENT_CO_FDC_Coupe_Fil_Droit) ]OTE(CO_Defaut_FDC);
   58: XIC(ENT_CO_Clef_Graissage)OTL(CO_Defaut_Clef_Graissage);
   59: XIO(ENT_CO_Clef_Graissage)XIC(CO_Acquit_defaut)OTU(CO_Defaut_Clef_Graissage);
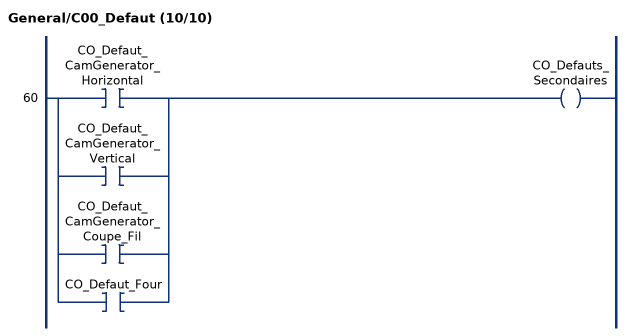
   60: [XIC(CO_Defaut_CamGenerator_Horizontal) ,XIC(CO_Defaut_CamGenerator_Vertical) ,XIC(CO_Defaut_CamGenerator_Coupe_Fil) ,XIC(CO_Defaut_Four) ]OTE(CO_Defauts_Secondaires);
END_ROUTINE
